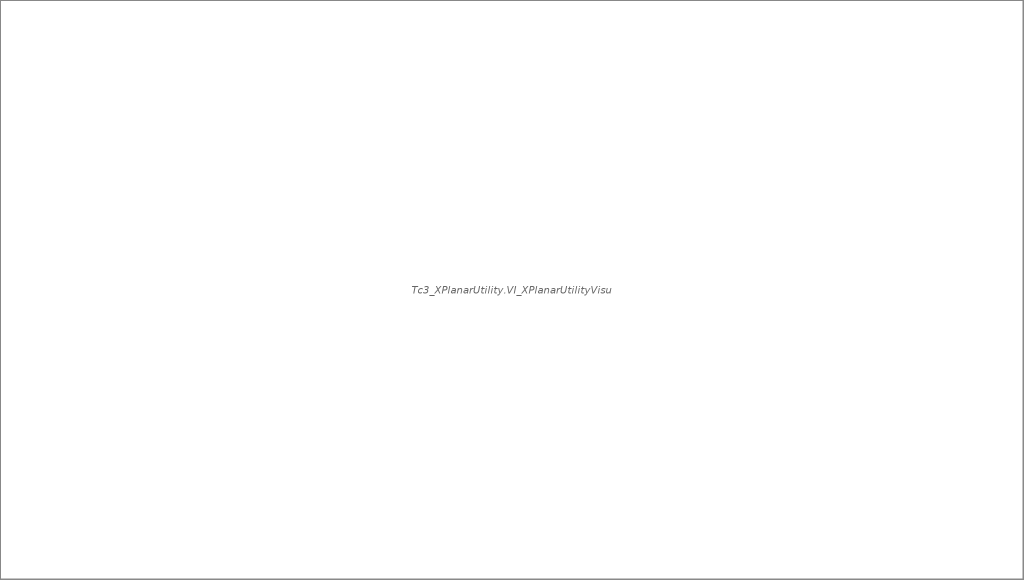
VISUALIZATION VI_Tc3_XPlanarUtility  // 1024x580
    Frame (0,0 1024x580)
        shows Tc3_XPlanarUtility.VI_XPlanarUtilityVisu()
END_VISUALIZATION

(* stored: Version 1.1.0.1
   Visu VI_Tc3_XPlanarUtility: Id {e462b8ef-95bc-4faf-86f6-08b5e31a7421} *)
